LIN {X 0,Y 119.789,Z 501.555,A -85,B 0,C 180,E1 -30604.131,E2 -30604.131} C_VEL
LIN {X 0,Y 119.842,Z 501.52,A -85,B 0,C 180,E1 -30604.468,E2 -30604.468} C_VEL
LIN {X 0,Y 109.394,Z 511.114,A -85,B 0,C 180,E1 -30605.248,E2 -30605.248} C_VEL
LIN {X 0,Y 98.98,Z 518.769,A -85,B 0,C 180,E1 -30606.237,E2 -30606.237} C_VEL
LIN {X 0,Y 88.602,Z 524.943,A -85,B 0,C 180,E1 -30607.464,E2 -30607.464} C_VEL
LIN {X 0,Y 78.296,Z 529.869,A -85,B 0,C 180,E1 -30609.104,E2 -30609.104} C_VEL
LIN {X 0,Y 68.091,Z 533.692,A -85,B 0,C 180,E1 -30611.312,E2 -30611.312} C_VEL
LIN {X 0,Y 58.055,Z 536.52,A -85,B 0,C 180,E1 -30614.42,E2 -30614.42} C_VEL
LIN {X 0,Y 45.07,Z 538.846,A -85,B 0,C 180,E1 -30620.667,E2 -30620.667} C_VEL
LIN {X 0,Y 38.876,Z 539.436,A -85,B 0,C 180,E1 -30625.316,E2 -30625.316} C_VEL
LIN {X 0,Y 33.034,Z 539.607,A -85,B 0,C 180,E1 -30631.673,E2 -30631.673} C_VEL
LIN {X 0,Y 23.616,Z 538.809,A -85,B 0,C 180,E1 -30653.467,E2 -30653.467} C_VEL
LIN {X 0,Y 20.887,Z 537.838,A -85,B 0,C 180,E1 -30670.331,E2 -30670.331} C_VEL
LIN {X 0,Y 20.183,Z 536.437,A -85,B 0,C 180,E1 -30689.993,E2 -30689.993} C_VEL
LIN {X 0,Y 21.937,Z 533.433,A -85,B 0,C 180,E1 -30718.715,E2 -30718.715} C_VEL
LIN {X 0,Y 27.671,Z 529.342,A -85,B 0,C 180,E1 -30739.628,E2 -30739.628} C_VEL
LIN {X 0,Y 37.196,Z 523.05,A -85,B 0,C 180,E1 -30753.822,E2 -30753.822} C_VEL
LIN {X 0,Y 46.184,Z 516.344,A -85,B 0,C 180,E1 -30761.073,E2 -30761.073} C_VEL
LIN {X 0,Y 52.644,Z 510.804,A -85,B 0,C 180,E1 -30764.679,E2 -30764.679} C_VEL
LIN {X 0,Y 61.063,Z 502.486,A -85,B 0,C 180,E1 -30768.029,E2 -30768.029} C_VEL
LIN {X 0,Y 69.475,Z 492.517,A -85,B 0,C 180,E1 -30770.488,E2 -30770.488} C_VEL
LIN {X 0,Y 76.274,Z 482.7,A -85,B 0,C 180,E1 -30772.089,E2 -30772.089} C_VEL
LIN {X 0,Y 82.286,Z 472.085,A -85,B 0,C 180,E1 -30773.143,E2 -30773.143} C_VEL
LIN {X 0,Y 87.018,Z 461.544,A -85,B 0,C 180,E1 -30773.904,E2 -30773.904} C_VEL
LIN {X 0,Y 91.377,Z 448.526,A -85,B 0,C 180,E1 -30774.553,E2 -30774.553} C_VEL
LIN {X 0,Y 94.193,Z 435.965,A -85,B 0,C 180,E1 -30775.032,E2 -30775.032} C_VEL
LIN {X 0,Y 95.688,Z 424.736,A -85,B 0,C 180,E1 -30775.378,E2 -30775.378} C_VEL
LIN {X 0,Y 95.112,Z 421.884,A -85,B 0,C 180,E1 -30779.47,E2 -30779.47} C_VEL
LIN {X 0,Y 94.957,Z 420.401,A -85,B 0,C 180,E1 -30782.12,E2 -30782.12} C_VEL
LIN {X 0,Y 94.903,Z 420.54,A -85,B 0,C 180,E1 -30787.981,E2 -30787.981} C_VEL
LIN {X 0,Y 95.417,Z 423.724,A -85,B 0,C 180,E1 -30793.716,E2 -30793.716} C_VEL
LIN {X 0,Y 95.666,Z 424.786,A -85,B 0,C 180,E1 -30795.157,E2 -30795.157} C_VEL
LIN {X 0,Y 93.583,Z 438.784,A -85,B 0,C 180,E1 -30795.665,E2 -30795.665} C_VEL
LIN {X 0,Y 90.532,Z 450.909,A -85,B 0,C 180,E1 -30796.344,E2 -30796.344} C_VEL
LIN {X 0,Y 86.414,Z 462.365,A -85,B 0,C 180,E1 -30797.141,E2 -30797.141} C_VEL
LIN {X 0,Y 81.325,Z 473.176,A -85,B 0,C 180,E1 -30798.09,E2 -30798.09} C_VEL
LIN {X 0,Y 74.552,Z 484.542,A -85,B 0,C 180,E1 -30799.498,E2 -30799.498} C_VEL
LIN {X 0,Y 67.061,Z 494.759,A -85,B 0,C 180,E1 -30801.556,E2 -30801.556} C_VEL
LIN {X 0,Y 59.621,Z 503.133,A -85,B 0,C 180,E1 -30804.005,E2 -30804.005} C_VEL
LIN {X 0,Y 49.942,Z 512.205,A -85,B 0,C 180,E1 -30808.423,E2 -30808.423} C_VEL
LIN {X 0,Y 40.684,Z 519.514,A -85,B 0,C 180,E1 -30814.867,E2 -30814.867} C_VEL
LIN {X 0,Y 33.465,Z 524.472,A -85,B 0,C 180,E1 -30822.696,E2 -30822.696} C_VEL
LIN {X 0,Y 31.139,Z 525.979,A -85,B 0,C 180,E1 -30826.161,E2 -30826.161} C_VEL
LIN {X 0,Y 26.869,Z 528.462,A -85,B 0,C 180,E1 -30832.615,E2 -30832.615} C_VEL
LIN {X 0,Y 19.207,Z 531.889,A -85,B 0,C 180,E1 -30846.061,E2 -30846.061} C_VEL
LIN {X 0,Y 14.183,Z 534.18,A -85,B 0,C 180,E1 -30866.486,E2 -30866.486} C_VEL
LIN {X 0,Y 13.044,Z 535.616,A -85,B 0,C 180,E1 -30890.637,E2 -30890.637} C_VEL
LIN {X 0,Y 13.449,Z 536.01,A -85,B 0,C 180,E1 -30898.843,E2 -30898.843} C_VEL
LIN {X 0,Y 17.4,Z 537.407,A -85,B 0,C 180,E1 -30923.897,E2 -30923.897} C_VEL
LIN {X 0,Y 22.848,Z 538.231,A -85,B 0,C 180,E1 -30937.355,E2 -30937.355} C_VEL
LIN {X 0,Y 29.745,Z 538.666,A -85,B 0,C 180,E1 -30946.336,E2 -30946.336} C_VEL
LIN {X 0,Y 42.34,Z 538.294,A -85,B 0,C 180,E1 -30954.87,E2 -30954.87} C_VEL
LIN {X 0,Y 49.24,Z 537.473,A -85,B 0,C 180,E1 -30957.632,E2 -30957.632} C_VEL
LIN {X 0,Y 57.369,Z 536,A -85,B 0,C 180,E1 -30960.002,E2 -30960.002} C_VEL
LIN {X 0,Y 70.36,Z 532.471,A -85,B 0,C 180,E1 -30962.693,E2 -30962.693} C_VEL
LIN {X 0,Y 77.49,Z 529.852,A -85,B 0,C 180,E1 -30963.908,E2 -30963.908} C_VEL
LIN {X 0,Y 67.058,Z 533.612,A -85,B 0,C 180,E1 -30965.328,E2 -30965.328} C_VEL
LIN {X 0,Y 56.701,Z 536.381,A -85,B 0,C 180,E1 -30967.424,E2 -30967.424} C_VEL
LIN {X 0,Y 43.073,Z 538.65,A -85,B 0,C 180,E1 -30971.752,E2 -30971.752} C_VEL
LIN {X 0,Y 36.403,Z 539.196,A -85,B 0,C 180,E1 -30975.126,E2 -30975.126} C_VEL
LIN {X 0,Y 23.818,Z 539.089,A -85,B 0,C 180,E1 -30987.709,E2 -30987.709} C_VEL
LIN {X 0,Y 14.407,Z 537.472,A -85,B 0,C 180,E1 -31020.792,E2 -31020.792} C_VEL
LIN {X 0,Y 13.065,Z 536.016,A -85,B 0,C 180,E1 -31049.989,E2 -31049.989} C_VEL
LIN {X 0,Y 16.052,Z 532.952,A -85,B 0,C 180,E1 -31091.04,E2 -31091.04} C_VEL
LIN {X 0,Y 23.671,Z 528.793,A -85,B 0,C 180,E1 -31112.95,E2 -31112.95} C_VEL
LIN {X 0,Y 34.644,Z 522.433,A -85,B 0,C 180,E1 -31124.479,E2 -31124.479} C_VEL
LIN {X 0,Y 44.863,Z 515.266,A -85,B 0,C 180,E1 -31130.188,E2 -31130.188} C_VEL
LIN {X 0,Y 54.823,Z 506.756,A -85,B 0,C 180,E1 -31133.436,E2 -31133.436} C_VEL
LIN {X 0,Y 63.45,Z 497.8,A -85,B 0,C 180,E1 -31135.433,E2 -31135.433} C_VEL
LIN {X 0,Y 71.269,Z 487.96,A -85,B 0,C 180,E1 -31136.765,E2 -31136.765} C_VEL
LIN {X 0,Y 77.372,Z 478.609,A -85,B 0,C 180,E1 -31137.603,E2 -31137.603} C_VEL
LIN {X 0,Y 83.495,Z 467.016,A -85,B 0,C 180,E1 -31138.214,E2 -31138.214} C_VEL
LIN {X 0,Y 88.254,Z 455.071,A -85,B 0,C 180,E1 -31138.73,E2 -31138.73} C_VEL
LIN {X 0,Y 92.021,Z 441.733,A -85,B 0,C 180,E1 -31139.205,E2 -31139.205} C_VEL
LIN {X 0,Y 94.182,Z 429.268,A -85,B 0,C 180,E1 -31139.553,E2 -31139.553} C_VEL
LIN {X 0,Y 94.012,Z 427.399,A -85,B 0,C 180,E1 -31143.213,E2 -31143.213} C_VEL
LIN {X 0,Y 93.985,Z 427.582,A -85,B 0,C 180,E1 -31147.248,E2 -31147.248} C_VEL
LIN {X 0,Y 94.146,Z 429.424,A -85,B 0,C 180,E1 -31151.013,E2 -31151.013} C_VEL
LIN {X 0,Y 91.695,Z 442.84,A -85,B 0,C 180,E1 -31151.53,E2 -31151.53} C_VEL
LIN {X 0,Y 87.894,Z 455.797,A -85,B 0,C 180,E1 -31152.144,E2 -31152.144} C_VEL
LIN {X 0,Y 82.884,Z 467.849,A -85,B 0,C 180,E1 -31152.817,E2 -31152.817} C_VEL
LIN {X 0,Y 76.804,Z 479.063,A -85,B 0,C 180,E1 -31153.542,E2 -31153.542} C_VEL
LIN {X 0,Y 69.076,Z 490.443,A -85,B 0,C 180,E1 -31154.869,E2 -31154.869} C_VEL
LIN {X 0,Y 60.504,Z 500.497,A -85,B 0,C 180,E1 -31156.614,E2 -31156.614} C_VEL
LIN {X 0,Y 50.335,Z 510.2,A -85,B 0,C 180,E1 -31159.541,E2 -31159.541} C_VEL
LIN {X 0,Y 40.365,Z 517.944,A -85,B 0,C 180,E1 -31163.935,E2 -31163.935} C_VEL
LIN {X 0,Y 32.274,Z 523.235,A -85,B 0,C 180,E1 -31169.43,E2 -31169.43} C_VEL
LIN {X 0,Y 23.177,Z 528.376,A -85,B 0,C 180,E1 -31180.714,E2 -31180.714} C_VEL
LIN {X 0,Y 15.205,Z 532.754,A -85,B 0,C 180,E1 -31207.57,E2 -31207.57} C_VEL
LIN {X 0,Y 13.449,Z 536.01,A -85,B 0,C 180,E1 -31258.843,E2 -31258.843} C_VEL
LIN {X 0,Y 15.637,Z 537.171,A -85,B 0,C 180,E1 -31280.104,E2 -31280.104} C_VEL
LIN {X 0,Y 21.261,Z 538.367,A -85,B 0,C 180,E1 -31305.672,E2 -31305.672} C_VEL
LIN {X 0,Y 27.492,Z 538.867,A -85,B 0,C 180,E1 -31317.487,E2 -31317.487} C_VEL
LIN {X 0,Y 32.944,Z 538.959,A -85,B 0,C 180,E1 -31322.001,E2 -31322.001} C_VEL
LIN {X 0,Y 34.871,Z 538.923,A -85,B 0,C 180,E1 -31322.779,E2 -31322.779} C_VEL
LIN {X 0,Y 35.186,Z 538.923,A -85,B 0,C 180,E1 -31322.876,E2 -31322.876} C_VEL
LIN {X 0,Y 35.223,Z 538.945,A -85,B 0,C 180,E1 -31323.873,E2 -31323.873} C_VEL
LIN {X 0,Y 21.452,Z 538.782,A -85,B 0,C 180,E1 -31330.595,E2 -31330.595} C_VEL
LIN {X 0,Y 14.834,Z 538.139,A -85,B 0,C 180,E1 -31338.605,E2 -31338.605} C_VEL
LIN {X 0,Y 8.903,Z 537.089,A -85,B 0,C 180,E1 -31357.843,E2 -31357.843} C_VEL
LIN {X 0,Y 5.953,Z 535.596,A -85,B 0,C 180,E1 -31409.976,E2 -31409.976} C_VEL
LIN {X 0,Y 11.66,Z 532.47,A -85,B 0,C 180,E1 -31474.676,E2 -31474.676} C_VEL
LIN {X 0,Y 21.389,Z 528.245,A -85,B 0,C 180,E1 -31490.275,E2 -31490.275} C_VEL
LIN {X 0,Y 33.446,Z 521.813,A -85,B 0,C 180,E1 -31496.394,E2 -31496.394} C_VEL
LIN {X 0,Y 43.709,Z 514.919,A -85,B 0,C 180,E1 -31499.296,E2 -31499.296} C_VEL
LIN {X 0,Y 54.471,Z 505.918,A -85,B 0,C 180,E1 -31500.951,E2 -31500.951} C_VEL
LIN {X 0,Y 64.167,Z 495.86,A -85,B 0,C 180,E1 -31502.006,E2 -31502.006} C_VEL
LIN {X 0,Y 72.106,Z 485.598,A -85,B 0,C 180,E1 -31502.563,E2 -31502.563} C_VEL
LIN {X 0,Y 79.171,Z 474.178,A -85,B 0,C 180,E1 -31503.015,E2 -31503.015} C_VEL
LIN {X 0,Y 84.465,Z 463.342,A -85,B 0,C 180,E1 -31503.204,E2 -31503.204} C_VEL
LIN {X 0,Y 88.898,Z 451.452,A -85,B 0,C 180,E1 -31503.435,E2 -31503.435} C_VEL
LIN {X 0,Y 92.217,Z 438.515,A -85,B 0,C 180,E1 -31503.646,E2 -31503.646} C_VEL
LIN {X 0,Y 92.996,Z 434.391,A -85,B 0,C 180,E1 -31503.822,E2 -31503.822} C_VEL
LIN {X 0,Y 92.932,Z 434.732,A -85,B 0,C 180,E1 -31506.787,E2 -31506.787} C_VEL
LIN {X 0,Y 89.855,Z 448.096,A -85,B 0,C 180,E1 -31507.222,E2 -31507.222} C_VEL
LIN {X 0,Y 85.628,Z 460.441,A -85,B 0,C 180,E1 -31507.647,E2 -31507.647} C_VEL
LIN {X 0,Y 79.848,Z 472.816,A -85,B 0,C 180,E1 -31508.049,E2 -31508.049} C_VEL
LIN {X 0,Y 72.842,Z 484.343,A -85,B 0,C 180,E1 -31508.543,E2 -31508.543} C_VEL
LIN {X 0,Y 64.989,Z 494.701,A -85,B 0,C 180,E1 -31509.339,E2 -31509.339} C_VEL
LIN {X 0,Y 57.128,Z 503.184,A -85,B 0,C 180,E1 -31510.221,E2 -31510.221} C_VEL
LIN {X 0,Y 46.693,Z 512.354,A -85,B 0,C 180,E1 -31511.965,E2 -31511.965} C_VEL
LIN {X 0,Y 36.321,Z 519.727,A -85,B 0,C 180,E1 -31514.667,E2 -31514.667} C_VEL
LIN {X 0,Y 26.013,Z 525.656,A -85,B 0,C 180,E1 -31519.004,E2 -31519.004} C_VEL
LIN {X 0,Y 16.054,Z 530.329,A -85,B 0,C 180,E1 -31528.913,E2 -31528.913} C_VEL
LIN {X 0,Y 9.801,Z 532.897,A -85,B 0,C 180,E1 -31545.798,E2 -31545.798} C_VEL
LIN {X 0,Y 7.026,Z 536.098,A -85,B 0,C 180,E1 -31636.894,E2 -31636.894} C_VEL
LIN {X 0,Y 14.377,Z 537.77,A -85,B 0,C 180,E1 -31667.913,E2 -31667.913} C_VEL
LIN {X 0,Y 27.787,Z 538.92,A -85,B 0,C 180,E1 -31680.003,E2 -31680.003} C_VEL
LIN {X 0,Y 34.871,Z 538.923,A -85,B 0,C 180,E1 -31682.779,E2 -31682.779} C_VEL
LIN {X 0,Y 36.84,Z 540.923,A -85,B 0,C 180,E1 -31683.358,E2 -31683.358} C_VEL
LIN {X 0,Y 36.84,Z 600,A -85,B 0,C 180,E1 -31683.358,E2 -31683.358} C_VEL
LIN {X 0,Y 36.84,Z 600,A -85,B 0,C 180,E1 -31683.358,E2 -31683.358}

QRS_NEXT_CUT()

QRS_NEXT()
QRS_HOME()

END
